FUNCTION_BLOCK FB_WareHouseWithRobotMove EXTENDS FB_ObjectBase_V2 IMPLEMENTS IBasicElement
VAR_INPUT
    Robot     : REFERENCE TO FB_FanucRobot_Basic;
    WareHouse : REFERENCE TO FB_WareHouse;
   // Command   : ST_WareHouseWithRobotMove_Command;
    Info	  : st_AutoSixAxisWarehouseParameter;
	Stop	  : BOOL;
END_VAR
VAR_OUTPUT
  // Status : ST_WareHouseWithRobotMove_Status;
END_VAR
VAR
	_Abort		: BOOL;
	strStatus	: STRING;
	uiResumeStep : UINT;
	ClampA_WareHouseCoordinates : ST_WareHouseCoordinates;
    ClampB_WareHouseCoordinates : ST_WareHouseCoordinates;
	UseA 	: BOOL;
	UseB	: BOOL;
	TargetWarehouse : E_WareHouse;
	Get 	:BOOL;
	tonTimeout		:TON;
	tonRobotTimeout		:TON;
	_UniqueErrorCode :STRING;
	PreviousStrStatus : STRING;
	PreviousErrorCode : STRING;
END_VAR

SUPER^.A10_StateControl();
A00_BasicUnits();

ACTION A00_BasicUnits:
tonTimeout(PT:=T#25S);
tonRobotTimeout(PT:=T#300S);
ErrorID :=2400;
END_ACTION

METHOD M_CheckCommand : BOOL // True : Command is useful
VAR_INPUT
END_VAR
VAR
	
END_VAR
// Check command paremeter is correct

IF NOT Info.Warehouse_A AND NOT Info.Warehouse_B THEN
	strStatus:='Wrong command , No warehouse selected';
	M_CheckCommand:=FALSE;
	RETURN;
ELSIF  Info.Warehouse_A AND  Info.Warehouse_B THEN
	strStatus:='Wrong command , Both warehouses selected';
	M_CheckCommand:=FALSE;
	RETURN;
ELSIF	Info.Warehouse_A THEN
	TargetWarehouse:=E_WareHouse.WareHouseA;
ELSIF	Info.Warehouse_B THEN
	TargetWarehouse:=E_WareHouse.WareHouseB;
END_IF

IF Info.Get_A <> Info.Get_B THEN
	strStatus:='Wrong command ,GetA not match to GetB';
	M_CheckCommand:=FALSE;
	RETURN;
	ELSE
		
	Get :=Info.Get_A;
END_IF


CASE LREAL_TO_INT(Info.Layer_A) OF

1,2,3,4,5,6,7,8,9,10:
	//Normal
	// Layer A in correct range
	IF ((Info.Slide_A < 1) OR (Info.Slide_A > 20)) THEN
		strStatus := 'Command error : Clamp A target slide out of range';
		M_CheckCommand:=FALSE;
		RETURN;
	ELSE
		ClampA_WareHouseCoordinates.Layer:=LREAL_TO_INT(Info.Layer_A);
		ClampA_WareHouseCoordinates.Slide:=LREAL_TO_INT(Info.Slide_A);
   
		UseA:=TRUE;	
	END_IF
	
99:
	UseA:=FALSE;
ELSE
	 strStatus := 'Command error : Clamp A target layer out of range.';
	 M_CheckCommand:=FALSE;
	 RETURN;
END_CASE


CASE LREAL_TO_INT(Info.Layer_B) OF

1,2,3,4,5,6,7,8,9,10:
//Normal
	// Layer A in correct range
	IF ((Info.Slide_B < 1) OR (Info.Slide_B > 20)) THEN
		strStatus := 'Command error : Clamp B target slide out of range';
		M_CheckCommand:=FALSE;
		RETURN;
	ELSE
		ClampB_WareHouseCoordinates.Layer:=LREAL_TO_INT(Info.Layer_B);
		ClampB_WareHouseCoordinates.Slide:=LREAL_TO_INT(Info.Slide_B);
		UseB:=TRUE;	
	END_IF
	
99:
		UseB:=FALSE;
ELSE
	 strStatus := 'Command error : Clamp B target layer out of range.';
	 M_CheckCommand:=FALSE;
	 RETURN;
END_CASE


M_CheckCommand:=TRUE;
END_METHOD

METHOD M_CheckUnitsNotBusy : BOOL
VAR_INPUT
END_VAR
M_CheckUnitsNotBusy := true;
END_METHOD

METHOD M_CheckUnitsReady : BOOL
VAR_INPUT
END_VAR
M_CheckUnitsReady := true;
END_METHOD

METHOD  M_STATE_ABORTED
VAR_INPUT
END_VAR
ERROR :=TRUE;
Busy    := FALSE;
Aborted := TRUE;
Status := strStatus;
UniqueErrorCode:=_UniqueErrorCode;
IF NOT Execute THEN
	eSTATE:=STATE_RESETTING;
END_IF

IF Execute AND Reset THEN
	PreviousStrStatus := strStatus;
	PreviousErrorCode := _UniqueErrorCode;
	uiExecutingStep :=uiResumeStep;
	eSTATE:=STATE_EXECUTING;
END_IF
END_METHOD

METHOD  M_STATE_ABORTING
VAR_INPUT
END_VAR
CASE uiAbortingStep OF
	0 :
		uiAbortingStep:=9999;
		IF strStatus = PreviousStrStatus THEN
			_UniqueErrorCode :=PreviousErrorCode;
		END_IF
		_Abort :=FALSE;
	9999:	_AbortCompleted:=TRUE;
END_CASE

IF _AbortCompleted THEN	
	eSTATE :=STATE_ABORTED;
END_IF
END_METHOD

METHOD  M_STATE_DONE
VAR_INPUT
END_VAR
Busy := FALSE;
Done := TRUE;
IF NOT Execute THEN
    eState := STATE_RESETTING;
END_IF
END_METHOD

METHOD  M_STATE_DORMANT
VAR_INPUT
END_VAR
// Clear FB output
Busy            := FALSE;
Done            := FALSE;
Aborted         := FALSE;
Error           := FALSE;
ErrorID         := 0;
Status          := '';
_ResetCompleted := FALSE;
_Error          := FALSE;
_Executed       := FALSE;
strStatus :='No Error';
tonTimeout.IN :=FALSE;
tonRobotTimeout.IN :=FALSE;
uiExecutingStep :=uiResettingStep :=uiResumeStep :=0;
PreviousStrStatus			 :='';
PreviousErrorCode			 :='';

// Wait Execute command
IF Execute THEN
    eState := STATE_EXECUTING;
END_IF
END_METHOD

METHOD  M_STATE_ERROR
VAR_INPUT
END_VAR
ERROR   :=TRUE;
Busy	:=FALSE;
Status := strStatus;
UniqueErrorCode:=_UniqueErrorCode;
IF NOT Execute THEN	
eSTATE:=STATE_RESETTING;
END_IF
END_METHOD

METHOD  M_STATE_EXECUTING
VAR_INPUT
END_VAR
VAR_INST
	BoxReady_1st : BOOL;
	BoxReady_2nd : BOOL;  
    uiBothStep : UINT;
    ClampA_WareHouseCoordinates : ST_WareHouseCoordinates;
    ClampB_WareHouseCoordinates : ST_WareHouseCoordinates;
	

	
END_VAR
VAR
	
END_VAR
// Set Busy active edit by johnson
Busy := TRUE;
IF THIS^.Stop THEN // Pending the timeout when Stop signal occur
	tonTimeout.IN :=FALSE;
	tonRobotTimeout.IN :=FALSE;
END_IF
// Service Process
CASE uiExecutingStep OF
	0:
        // Clear variable
       
        tonTimeout.IN :=FALSE;
        uiBothStep := 0;
		BoxReady_1st := 0;
		BoxReady_2nd := 0;
        // Check command
        IF M_CheckCommand() THEN
            uiExecutingStep := 10;
		ELSE
			_Error:=TRUE;
        END_IF
    10:
        // Start process, check units first
        IF M_CheckUnitsReady() THEN
            uiExecutingStep := 20;
        END_IF
    20:
        // CHeck units not busy state
        IF M_CheckUnitsNotBusy() THEN
            uiExecutingStep := 1000;
        END_IF
   
	1000:   
			// Read  Warehouse coordinate
			ClampA_WareHouseCoordinates := THIS^.ClampA_WareHouseCoordinates;
            ClampB_WareHouseCoordinates := THIS^.ClampB_WareHouseCoordinates;     
			IF UseA AND NOT UseB THEN
				//Only clampA
				uiExecutingStep := 10000;
			ELSIF NOT UseA AND UseB THEN
				//Only ClampB 
				uiExecutingStep := 20000;
			ELSIF UseA AND UseB THEN
				//Both Clamps
				uiExecutingStep := 30000;		
			END_IF
       
    10000: // Only ClampA 
        IF NOT Robot._DI1.Done THEN
            // Read ClampA Warehouse coordinate
            ClampA_WareHouseCoordinates := THIS^.ClampA_WareHouseCoordinates;
			
			IF Get THEN// Prepare Box
				//Pick Box
				 WareHouse.M_StartReloadBox(WareHouseSelect := TargetWarehouse, WarehouseCoordinates := ClampA_WareHouseCoordinates);

           		 // Check Box reload completed
           		 IF WareHouse.bReloadBox_Completed THEN
           	     BoxReady_1st := TRUE;
          		  END_IF
				  // Robot Warehouse move
           		 Robot.M_StartWareHousePickUpBox_ClampA(WareHouseSelect := TargetWarehouse,
                                                   Info            := ClampA_WareHouseCoordinates,
                                                   BoxReady_1st    := BoxReady_1st);
				tonTimeout.IN:=TRUE;
				IF tonTimeout.Q THEN
					_Error:=TRUE;
					strStatus:='Clamp A reolad box timeout';
				END_IF
				  
			ELSE
					//Place Box
					WareHouse.M_StartFeedInBox(WareHouseSelect := TargetWarehouse, WarehouseCoordinates := ClampA_WareHouseCoordinates);

           			 // Check Box reload completed
           			 IF WareHouse.bFeedInBox_Completed THEN
               			 BoxReady_1st := TRUE;
          		 	 END_IF				
					           
			 	Robot.M_StartWareHousePlaceBox_ClampA(WareHouseSelect := TargetWarehouse,
                                                   Info            := ClampA_WareHouseCoordinates,
                                                   BoxReady_1st    := BoxReady_1st);
            	
				tonTimeout.IN:=TRUE;
				IF tonTimeout.Q THEN
					_Error:=TRUE;
					strStatus:='Clamp A Feedin box timeout';
				END_IF
           END_IF
        ELSE
            uiExecutingStep := 10080;
        END_IF
		
		tonRobotTimeout.IN :=TRUE;
		IF tonRobotTimeout.Q THEN
			_Error:=TRUE;
			strStatus:='Clamp A  robot timeout';
		END_IF
		
    10080:
        Robot.M_ResetAllCommand(); // Clear command and go to place box
		tonTimeout.IN :=FALSE;
		tonRobotTimeout.IN :=FALSE;
        IF NOT Robot._DI1.Done THEN
            uiExecutingStep := 99000; 
        END_IF
    
    
   20000: // Only ClampB
        IF NOT Robot._DI1.Done THEN
            			
			IF Get THEN// Prepare Box
				//Pick Box
				 WareHouse.M_StartReloadBox(WareHouseSelect := TargetWarehouse, WarehouseCoordinates := ClampB_WareHouseCoordinates);

           		 // Check Box reload completed
           		 IF WareHouse.bReloadBox_Completed THEN
           	     BoxReady_2nd := TRUE;
          		  END_IF
				  // Robot Warehouse move
           		 Robot.M_StartWareHousePickUpBox_ClampB(WareHouseSelect := TargetWarehouse,
                                                   Info            := ClampB_WareHouseCoordinates,
                                                   BoxReady_2nd    := BoxReady_2nd);

				tonTimeout.IN:=TRUE;
				IF tonTimeout.Q THEN
					_Error:=TRUE;
					strStatus:='Clamp B Reload box timeout';
				END_IF
			ELSE
					//Place Box
					WareHouse.M_StartFeedInBox(WareHouseSelect := TargetWarehouse, WarehouseCoordinates := ClampB_WareHouseCoordinates);

           			 // Check Box reload completed
           			 IF WareHouse.bFeedInBox_Completed THEN
               			 BoxReady_2nd := TRUE;
          		 	 END_IF				
					           
			 	Robot.M_StartWareHousePlaceBox_ClampB (WareHouseSelect := TargetWarehouse,
                                                   Info            := ClampB_WareHouseCoordinates,
                                                   BoxReady_2nd    := BoxReady_2nd);
            	tonTimeout.IN:=TRUE;
				IF tonTimeout.Q THEN
					_Error:=TRUE;
					strStatus:='Clamp B Feedin box timeout';
				END_IF
           END_IF
        ELSE
            uiExecutingStep := 20080;
        END_IF
		tonRobotTimeout.IN :=TRUE;
		IF tonRobotTimeout.Q THEN
			_Error:=TRUE;
			strStatus:='Clamp B Robot timeout';
		END_IF
		
    20080:
        Robot.M_ResetAllCommand(); // Clear command and go to place box
		tonTimeout.IN :=FALSE;
		tonRobotTimeout.IN :=FALSE;

        IF NOT Robot._DI1.Done THEN
            uiExecutingStep := 99000; 
        END_IF
		
    30000: // Both Clamps
        		
		IF Get THEN //BOth clamps pick
        CASE uiBothStep OF
            0: // ClampA target slide move the box to front side
                WareHouse.M_StartReloadBox(WareHouseSelect      := TargetWarehouse,
                                           WarehouseCoordinates := ClampA_WareHouseCoordinates);
				
				tonTimeout.IN :=TRUE;
				IF tonTimeout.Q THEN
					_Error:=TRUE;
					strStatus:='Clamp A reload timeout';
				END_IF
               
                IF WareHouse.bReloadBox_Completed THEN
					tonTimeout.IN :=FALSE;
                    BoxReady_1st     := TRUE;
                    uiBothStep := 10;
                END_IF

            10: // wait Robot Allow continue
			 		WareHouse.M_ResetReloadBox();
                IF Robot._DI1.Notification // AND
//                    NOT
//                    WareHouse._stWarehouseList.ASide_Layers[ClampA_WareHouseCoordinates.Layer].stStatus.bSlides[ClampA_WareHouseCoordinates.Slide]
                    THEN
                   
					
                    IF NOT WareHouse.bReloadBox_Completed THEN					
               
                        uiBothStep := 15;
                    END_IF

                END_IF
			15:	IF NOT WareHouse._stWarehouseList.ASide_Layers[ClampA_WareHouseCoordinates.Layer].stStatus.bSlides[ClampA_WareHouseCoordinates.Slide] THEN
					 uiBothStep := 20;	
				 END_IF
				 
            20: // ClampB target slide move the box to front slide
                WareHouse.M_StartReloadBox(WareHouseSelect := TargetWarehouse, WarehouseCoordinates := ClampB_WareHouseCoordinates);
				tonTimeout.IN :=TRUE;
                IF WareHouse.bReloadBox_Completed THEN
					tonTimeout.IN :=FALSE;
                    BoxReady_2nd     := TRUE;
                    uiBothStep := 99;
                END_IF
				IF tonTimeout.Q THEN
					_Error:=TRUE;
					strStatus:='Clamp B reload timeout';
				END_IF
				
				
            99:
				WareHouse.M_ResetReloadBox();
        // wait reset
        END_CASE

        Robot.M_StartWareHousePickUpBox_ClampBoth(WareHouseSelect := TargetWarehouse,
                                                  ClampA_Info     := ClampA_WareHouseCoordinates,
                                                  ClampB_Info     := ClampB_WareHouseCoordinates,
                                                  BoxReady_1st    := BoxReady_1st,
                                                  BoxReady_2nd    := BoxReady_2nd);
												  
		tonRobotTimeout.IN :=TRUE;
		IF tonRobotTimeout.Q THEN
			_Error:=TRUE;
			strStatus:='Robot timeout';
		END_IF
		ELSE
		  CASE uiBothStep OF
			  
			   0: // ClampA target slide move the box to front side
                WareHouse.M_StartFeedInBox(WareHouseSelect      := TargetWarehouse,
                                           WarehouseCoordinates := ClampA_WareHouseCoordinates);

               tonTimeout.IN :=TRUE;
                IF WareHouse.bFeedInBox_Completed THEN
					tonTimeout.IN :=FALSE;
                    BoxReady_1st     := TRUE;
                    uiBothStep := 10;
                END_IF
				IF tonTimeout.Q THEN
					_Error:=TRUE;
					strStatus:='Clamp A Feedin timeout';
				END_IF

            10: // wait Robot Allow continue
					WareHouse.M_ResetFeedInBox();
                 IF Robot._DI1.Notification //AND
                     
//                    WareHouse._stWarehouseList.ASide_Layers[ClampA_WareHouseCoordinates.Layer].stStatus.bSlides[ClampA_WareHouseCoordinates.Slide]
                    THEN
                    

                    IF NOT WareHouse.bFeedInBox_Completed THEN
                        uiBothStep := 15;
                    END_IF

                END_IF
			15:  
				uiBothStep := 20;
			
            20: // ClampB target slide move the box to front slide
                WareHouse.M_StartFeedInBox(WareHouseSelect := TargetWarehouse, WarehouseCoordinates := ClampB_WareHouseCoordinates);
				tonTimeout.IN :=TRUE;
                IF WareHouse.bFeedInBox_Completed THEN
					tonTimeout.IN :=FALSE;
                    BoxReady_2nd     := TRUE;
                    uiBothStep := 99;
                END_IF
				IF tonTimeout.Q THEN
					_Error:=TRUE;
					strStatus:='Clamp B Feedin timeout';
				END_IF
            99: 
				WareHouse.M_ResetFeedInBox();

        END_CASE

        Robot.M_StartWareHousePlaceUpBox_ClampBoth(WareHouseSelect := TargetWarehouse,
                                                  ClampA_Info     := ClampA_WareHouseCoordinates,
                                                  ClampB_Info     := ClampB_WareHouseCoordinates,
                                                  BoxReady_1st    := BoxReady_1st,
                                                  BoxReady_2nd    := BoxReady_2nd);
												  
		tonRobotTimeout.IN :=TRUE;
		IF tonRobotTimeout.Q THEN
			_Error:=TRUE;
			strStatus:='Robot timeout';
		END_IF
		END_IF
		
        IF Robot._DI1.Done THEN
            uiExecutingStep := 30080;
        END_IF
		
    30080: // Check robot command is clear
        WareHouse.M_ResetReloadBox();
        WareHouse.M_ResetFeedInBox();
        Robot.M_ResetAllCommand();
		tonTimeout.IN :=FALSE;
		tonRobotTimeout.IN :=FALSE;
		
        IF NOT Robot._DI1.Done THEN
            uiExecutingStep := 99000; // go to place step
        END_IF    
   
   
    99000: // process done
                Status    := 'Process completed';
        _Executed := TRUE;
END_CASE
IF _Executed THEN
    eState := STATE_DONE;
ELSIF _Error THEN
	//FUN_UniqueErrorCodeGenerator(iErrorID := ErrorID,UinqueErrorCode=>_UniqueErrorCode);
    eState := STATE_ERROR;
ELSIF NOT Execute THEN
    eState := STATE_RESETTING;
END_IF
IF _Abort OR Abort THEN
	//FUN_UniqueErrorCodeGenerator(iErrorID := ErrorID,UinqueErrorCode=>_UniqueErrorCode);
	eSTATE:=STATE_ABORTING;
END_IF
END_METHOD

METHOD  M_STATE_RESETTING
VAR_INPUT
END_VAR
Error :=FALSE;
Done :=FALSE;
Busy := FALSE;
_Error :=FALSE;

CASE uiResettingStep OF
	
	0:
		tonTimeout.IN :=FALSE;
		Robot.M_ResetAllCommand();
		uiResettingStep:=9999;
		WareHouse.M_ResetFeedInBox();
		WareHouse.M_ResetReloadBox();
	9999:
		_ResetCompleted:=TRUE;
END_CASE
IF _ResetCompleted THEN
	eSTATE:=STATE_DORMANT;
END_IF
END_METHOD

END_FUNCTION_BLOCK

(* stored: Version 1.1.0.1, ProductVersion 3.1.4024.13
   POU FB_WareHouseWithRobotMove: Id {c34f18a3-22c7-4de8-baa3-1fa49642345b}, SpecialFunc None
   Folder Method: Id {89696213-4019-4c9c-9f67-931f10b5f345}
   Folder State: Id {5de75564-90d9-4f04-b2b4-8beaf8aee9f2}
   Action A00_BasicUnits: Id {0a9d1eb2-ece8-4258-868d-9fca98379a85}
   Method M_CheckCommand: Id {a76b766b-4e58-4d01-b36b-ac9e3c19bef8}
   Method M_CheckUnitsNotBusy: Id {5b2a2e93-dc01-4672-9dcc-d2bde62d5696}
   Method M_CheckUnitsReady: Id {b768fa53-75be-4c0f-b659-de7fa315ef9f}
   Method M_STATE_ABORTED: Id {32cc8b5c-bf2e-497c-914f-04ec1622ac0f}
   Method M_STATE_ABORTING: Id {8f6fb6a4-324c-4a1e-8128-e31260951494}
   Method M_STATE_DONE: Id {46561604-3447-4214-9357-599c811963ec}
   Method M_STATE_DORMANT: Id {ee4597f2-2dea-496b-8045-5fcc940e1c57}
   Method M_STATE_ERROR: Id {df32d5ac-f837-4572-919b-783d09fef90d}
   Method M_STATE_EXECUTING: Id {c8d7c663-589c-412d-b2ca-18dec4dcd426}
   Method M_STATE_RESETTING: Id {8d7a6c7f-081f-440a-bece-0e01213ed74e} *)
